(* IEC 61131-3 sources: eCockpitGit/test_project/src/%F%00 Library/%F%Common Functions/%F%Buffer/%POU%FB_FIFOQueue, 7 files *)

(* ---- %METH%peek.st ---- *)
//Gets the oldest element from the buffer if there are any, without removing it from the buffer
// |**Version**|**Author**| **Date** |**Changes**
// | 1         | NSN      | 15-02-22 | Creation
METHOD peek : BOOL
VAR_INPUT
	value		:ANY;
END_VAR

(*%!%__DELIMITER__%!%*)
peek			:=		peekManuel(valuePoint:=value.pValue,valueSize:=TO_DWORD(value.diSize));

(* ---- %METH%peekManuel.st ---- *)
//Gets the oldest element from the buffer if there are any, without removing it from the buffer
// |**Version**|**Author**| **Date** |**Changes**
// | 1         | NSN      | 15-02-22 | Creation
METHOD peekManuel : BOOL
VAR_INPUT
	valuePoint	:POINTER TO BYTE;
	valueSize	:DWORD;
END_VAR
VAR
	i			:DWORD;
	position	:DWORD;
	buffer		:POINTER TO BYTE;
	trans		:DWORD;
END_VAR
(*%!%__DELIMITER__%!%*)
WHILE S_amount > 0 DO
	IF __COMPARE_AND_SWAP(ADR(S_blockOutput),0,1) THEN
		IF S_amount = 0 THEN
			S_blockOutput			:=		0;
			RETURN;
		END_IF
		IF S_output < S_bufferSize THEN
			position				:=		S_output + 1;
		ELSE
			position				:=		0;
		END_IF
		buffer						:=		S_buffer + (S_elementSize * position);
		trans						:=		MIN(valueSize,S_elementSize);
		FOR i := 1 TO trans DO
			IF i > valueSize THEN
				valuePoint^			:=		0;
			ELSE
				valuePoint^			:=		buffer^;
			END_IF
			buffer					:=		buffer + 1;
			valuePoint				:=		valuePoint + 1;
		END_FOR
		peekManuel					:=		TRUE;
		S_blockOutput				:=		0;
		RETURN;
	END_IF
END_WHILE

(* ---- %METH%push.st ---- *)
//Pushes the given element to the queue
// |**Version**|**Author**| **Date** |**Changes**
// | 1         | NSN      | 15-02-22 | Creation
METHOD push : BOOL
VAR_INPUT
	value		:ANY;
END_VAR
(*%!%__DELIMITER__%!%*)
push		:=		pushManuel(valuePoint:=value.pValue,valueSize:=TO_DWORD(value.diSize));

(* ---- %METH%pushManuel.st ---- *)
//Pushes the given element to the queue
// |**Version**|**Author**| **Date** |**Changes**
// | 1         | NSN      | 15-02-22 | Creation
METHOD pushManuel : BOOL
VAR_INPUT
	valuePoint	:POINTER TO BYTE;
	valueSize	:DWORD;
END_VAR
VAR
	i			:DWORD;
	buffer		:POINTER TO BYTE;
END_VAR
(*%!%__DELIMITER__%!%*)
WHILE S_amount < S_bufferSize DO
	IF __COMPARE_AND_SWAP(ADR(S_blockInput),0,1) THEN
		IF S_amount = S_bufferSize THEN
			S_blockInput			:=		0;
			RETURN;
		END_IF
		IF S_input < S_bufferSize - 1 THEN
			S_input					:=		S_input + 1;
		ELSE
			S_input					:=		0;
		END_IF
		buffer						:=		S_buffer + (S_elementSize * S_input);
		FOR i := 1 TO S_elementSize DO
			IF i > valueSize THEN
				buffer^				:=		0;
			ELSE
				buffer^				:=		valuePoint^;
			END_IF
			buffer					:=		buffer + 1;
			valuePoint				:=		valuePoint + 1;
		END_FOR
		WHILE TRUE DO
			IF __COMPARE_AND_SWAP(ADR(S_block),0,1) THEN
				S_amount			:=		S_amount + 1;
				S_block				:=		0;
				EXIT;
			END_IF
		END_WHILE

		pushManuel					:=		TRUE;
		S_blockInput				:=		0;
		RETURN;
	END_IF
END_WHILE

(* ---- %METH%setSize.st ---- *)
//Changes the size of the queue in a tread safe way
// |**Version**|**Author**| **Date** |**Changes**
// | 1         | NSN      | 15-02-22 | Creation
METHOD setSize
VAR_INPUT
	size		:DWORD;
END_VAR

(*%!%__DELIMITER__%!%*)
WHILE TRUE DO
	IF __COMPARE_AND_SWAP(ADR(S_block),0,1) THEN
		S_bufferSize					:=		size;
		S_amount				:=		0;
		S_input					:=		0;
		S_output				:=		0;
		S_block					:=		0;
		RETURN;
	END_IF
END_WHILE

(* ---- %METH%unshift.st ---- *)
//Gets the oldest element from the buffer if there are any
// |**Version**|**Author**| **Date** |**Changes**
// | 1         | NSN      | 15-02-22 | Creation
METHOD unshift : BOOL
VAR_INPUT
	value		:ANY;
END_VAR

(*%!%__DELIMITER__%!%*)
unshift			:=		unshiftManuel(valuePoint:=value.pValue,valueSize:=TO_DWORD(value.diSize));

(* ---- %METH%unshiftManuel.st ---- *)
//Gets the oldest element from the buffer if there are any
// |**Version**|**Author**| **Date** |**Changes**
// | 1         | NSN      | 15-02-22 | Creation
METHOD unshiftManuel : BOOL
VAR_INPUT
	valuePoint	:POINTER TO BYTE;
	valueSize	:DWORD;
END_VAR
VAR
	i			:DWORD;
	buffer		:POINTER TO BYTE;
	trans		:DWORD;
END_VAR
(*%!%__DELIMITER__%!%*)
WHILE S_amount > 0 DO
	IF __COMPARE_AND_SWAP(ADR(S_blockOutput),0,1) THEN
		IF S_amount = 0 THEN
			S_blockOutput			:=		0;
			RETURN;
		END_IF
		IF S_output < S_bufferSize - 1 THEN
			S_output				:=		S_output + 1;
		ELSE
			S_output				:=		0;
		END_IF
		buffer						:=		S_buffer + (S_elementSize * S_output);
		trans						:=		MIN(valueSize,S_elementSize);
		FOR i := 1 TO trans DO
			IF i > valueSize THEN
				valuePoint^			:=		0;
			ELSE
				valuePoint^			:=		buffer^;
			END_IF
			buffer					:=		buffer + 1;
			valuePoint				:=		valuePoint + 1;
		END_FOR
		WHILE TRUE DO
			IF __COMPARE_AND_SWAP(ADR(S_block),0,1) THEN
				S_amount			:=		S_amount - 1;
				S_block				:=		0;
				EXIT;
			END_IF
		END_WHILE

		unshiftManuel				:=		TRUE;
		S_blockOutput				:=		0;
		RETURN;
	END_IF
END_WHILE
